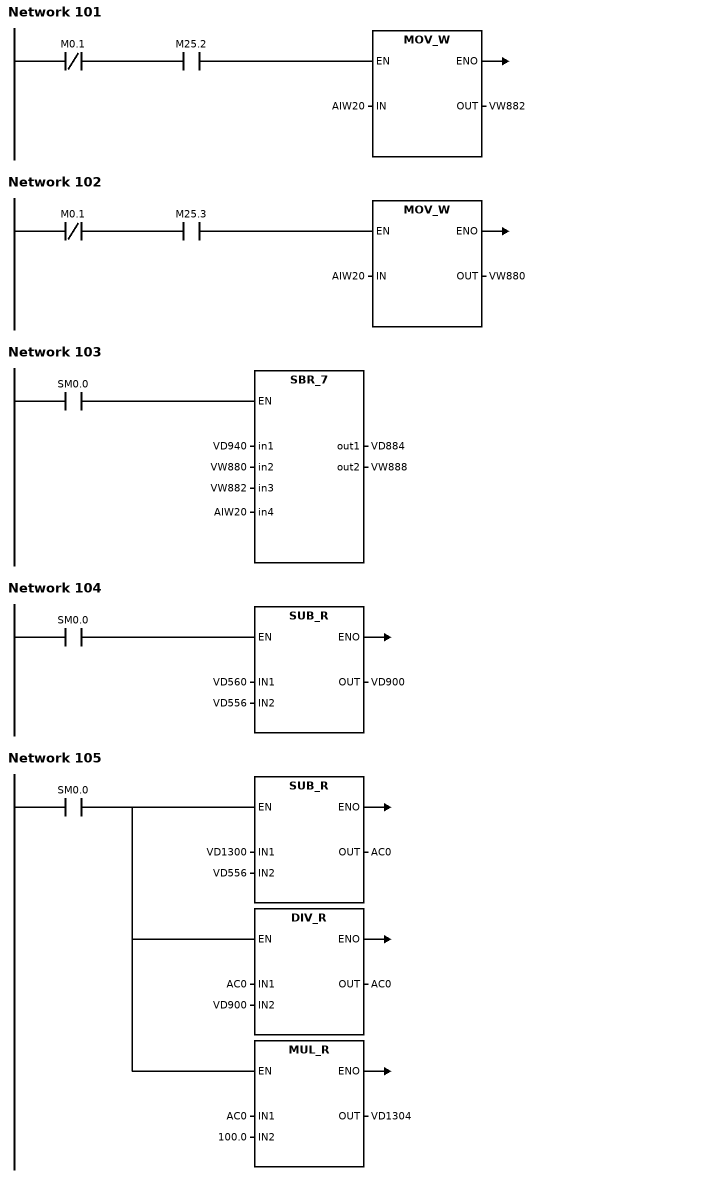
[picture p24: OB1 networks 101-105]
Network 101
LDN    M0.1
A      M25.2
MOVW   AIW20, VW882
Network 102
LDN    M0.1
A      M25.3
MOVW   AIW20, VW880
Network 103
LD     SM0.0
CALL   SBR_7:SBR7, VD940, VW880, VW882, AIW20, VD884, VW888
Network 104
LD     SM0.0
MOVR   VD560, VD900
-R     VD556, VD900
Network 105
LD     SM0.0
MOVR   VD1300, AC0
-R     VD556, AC0
/R     VD900, AC0
MOVR   AC0, VD1304
*R     100.0, VD1304
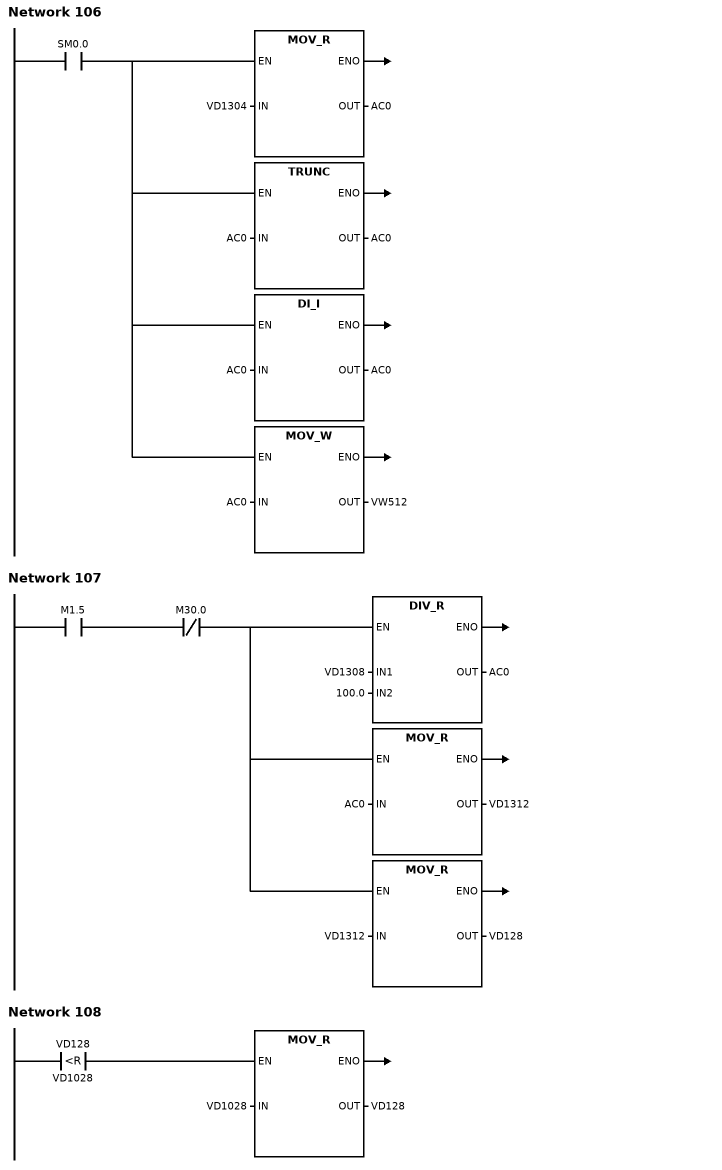
Network 106
LD     SM0.0
MOVR   VD1304, AC0
TRUNC  AC0, AC0
DTI    AC0, AC0
MOVW   AC0, VW512
Network 107
LD     M1.5
AN     M30.0
MOVR   VD1308, AC0
/R     100.0, AC0
MOVR   AC0, VD1312
MOVR   VD1312, VD128
Network 108
LDR<   VD128, VD1028
MOVR   VD1028, VD128
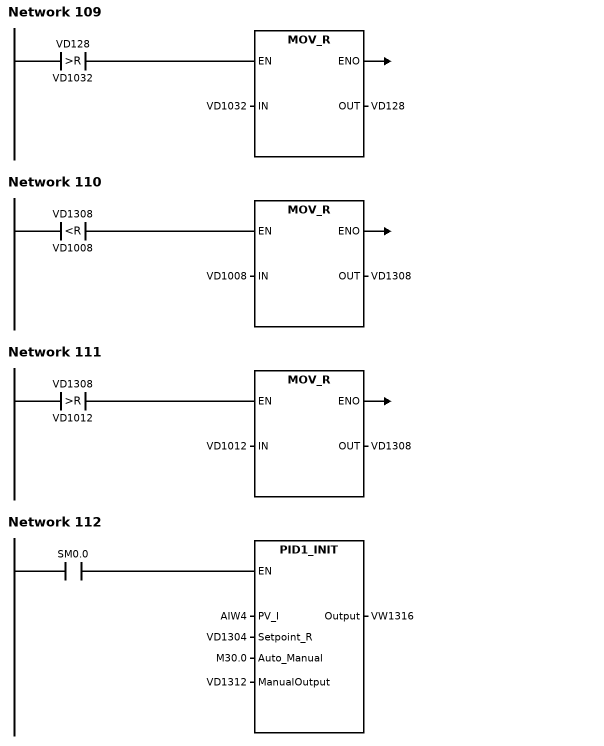
Network 109
LDR>   VD128, VD1032
MOVR   VD1032, VD128
Network 110
LDR<   VD1308, VD1008
MOVR   VD1008, VD1308
Network 111
LDR>   VD1308, VD1012
MOVR   VD1012, VD1308
Network 112
LD     SM0.0
CALL   PID1_INIT:SBR2, AIW4, VD1304, M30.0, VD1312, VW1316
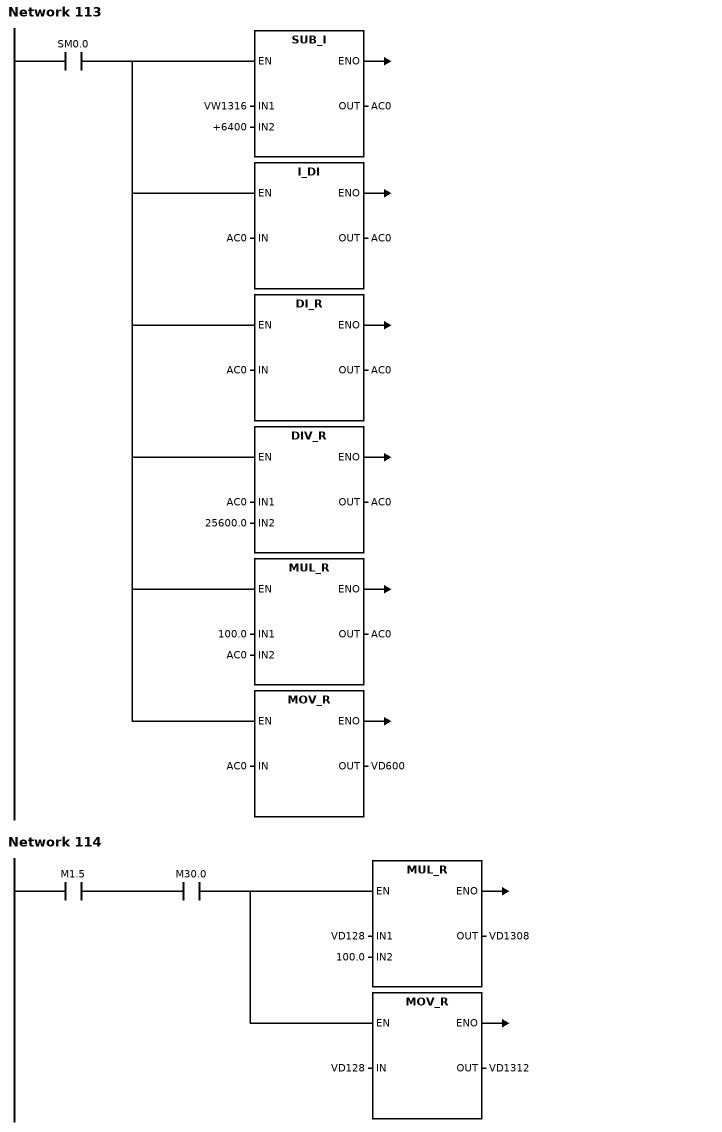
Network 113
LD     SM0.0
MOVW   VW1316, AC0
-I     +6400, AC0
ITD    AC0, AC0
DTR    AC0, AC0
/R     25600.0, AC0
*R     100.0, AC0
MOVR   AC0, VD600
Network 114
LD     M1.5
A      M30.0
MOVR   VD128, VD1308
*R     100.0, VD1308
MOVR   VD128, VD1312
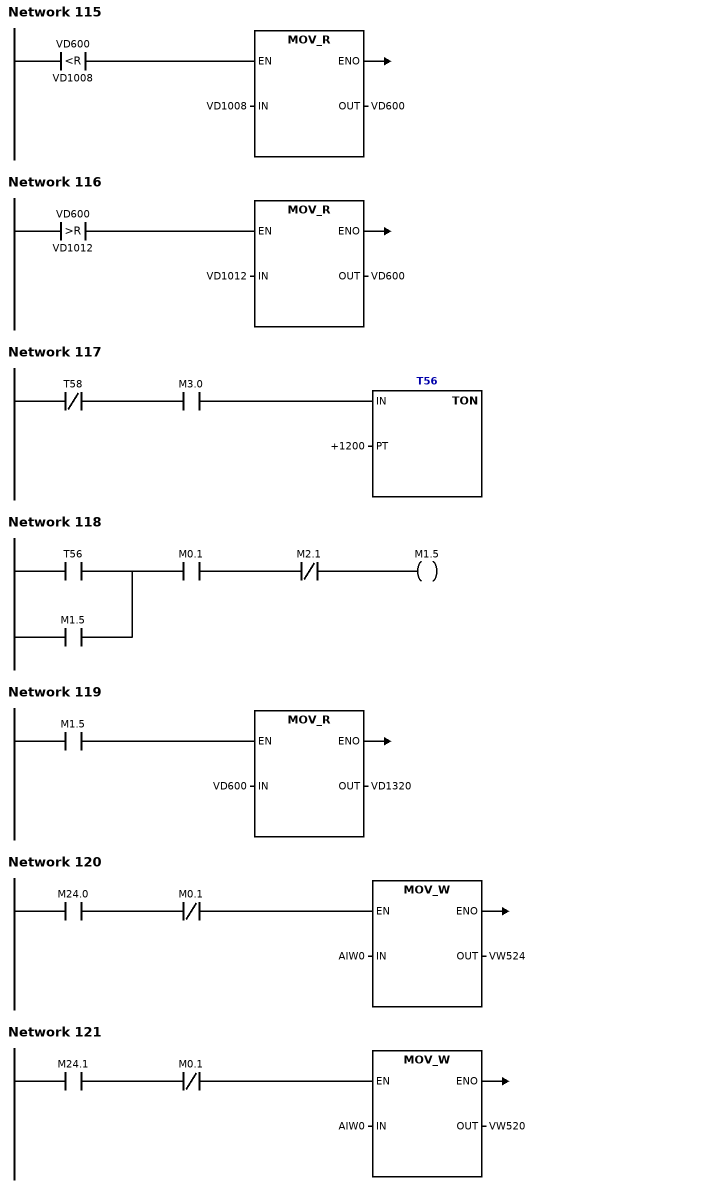
Network 115
LDR<   VD600, VD1008
MOVR   VD1008, VD600
Network 116
LDR>   VD600, VD1012
MOVR   VD1012, VD600
Network 117
LDN    T58
A      M3.0
TON    T56, +1200
Network 118
LD     T56
O      M1.5
A      M0.1
AN     M2.1
=      M1.5
Network 119
LD     M1.5
MOVR   VD600, VD1320
Network 120
LD     M24.0
AN     M0.1
MOVW   AIW0, VW524
Network 121
LD     M24.1
AN     M0.1
MOVW   AIW0, VW520
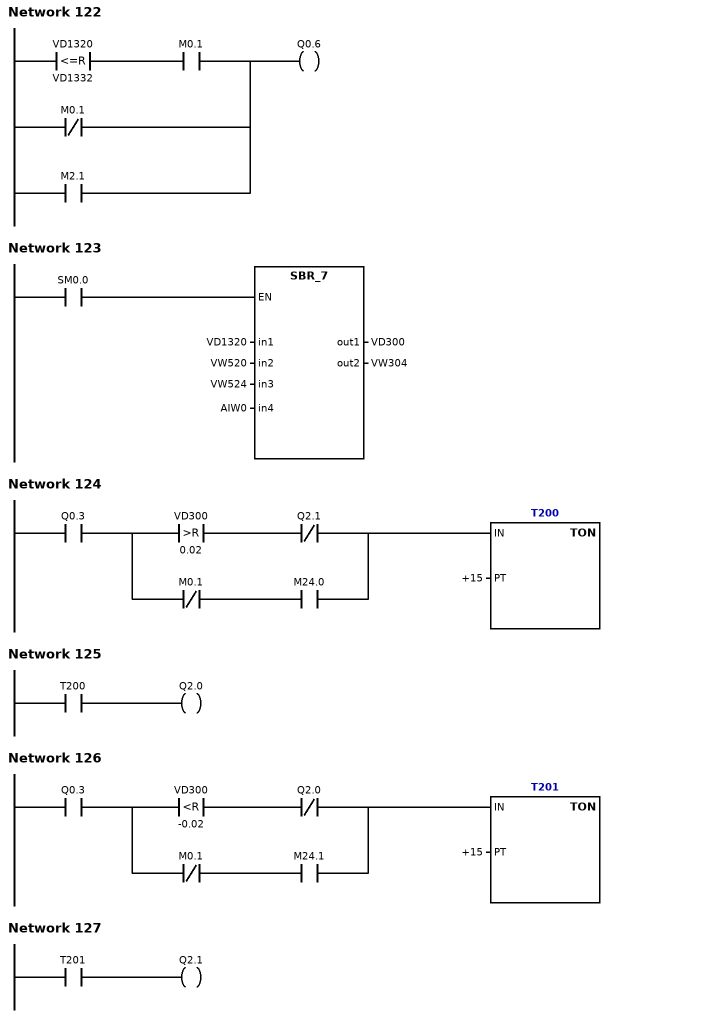
Network 122
LDR<=  VD1320, VD1332
A      M0.1
ON     M0.1
O      M2.1
=      Q0.6
Network 123
LD     SM0.0
CALL   SBR_7:SBR7, VD1320, VW520, VW524, AIW0, VD300, VW304
Network 124
LD     Q0.3
LDR>   VD300, 0.02
AN     Q2.1
LDN    M0.1
A      M24.0
OLD
ALD
TON    T200, +15
Network 125
LD     T200
=      Q2.0
Network 126
LD     Q0.3
LDR<   VD300, -0.02
AN     Q2.0
LDN    M0.1
A      M24.1
OLD
ALD
TON    T201, +15
Network 127
LD     T201
=      Q2.1
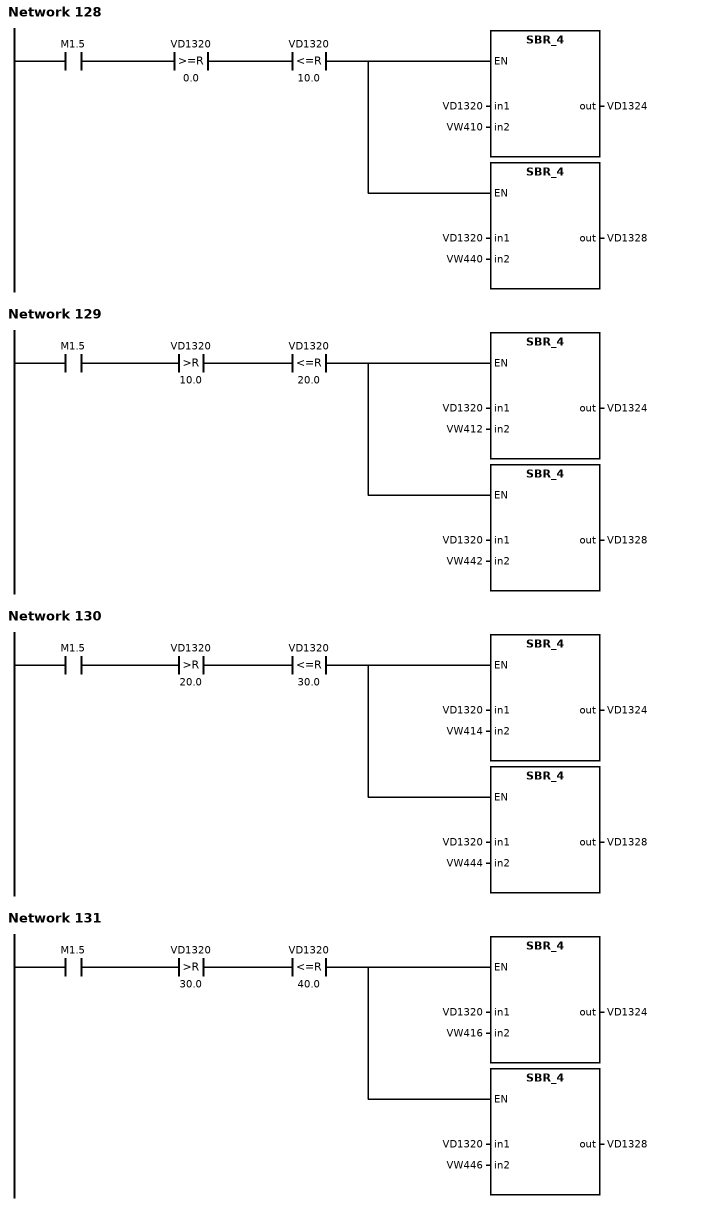
Network 128
LD     M1.5
AR>=   VD1320, 0.0
AR<=   VD1320, 10.0
CALL   SBR_4:SBR4, VD1320, VW410, VD1324
CALL   SBR_4:SBR4, VD1320, VW440, VD1328
Network 129
LD     M1.5
AR>    VD1320, 10.0
AR<=   VD1320, 20.0
CALL   SBR_4:SBR4, VD1320, VW412, VD1324
CALL   SBR_4:SBR4, VD1320, VW442, VD1328
Network 130
LD     M1.5
AR>    VD1320, 20.0
AR<=   VD1320, 30.0
CALL   SBR_4:SBR4, VD1320, VW414, VD1324
CALL   SBR_4:SBR4, VD1320, VW444, VD1328
Network 131
LD     M1.5
AR>    VD1320, 30.0
AR<=   VD1320, 40.0
CALL   SBR_4:SBR4, VD1320, VW416, VD1324
CALL   SBR_4:SBR4, VD1320, VW446, VD1328
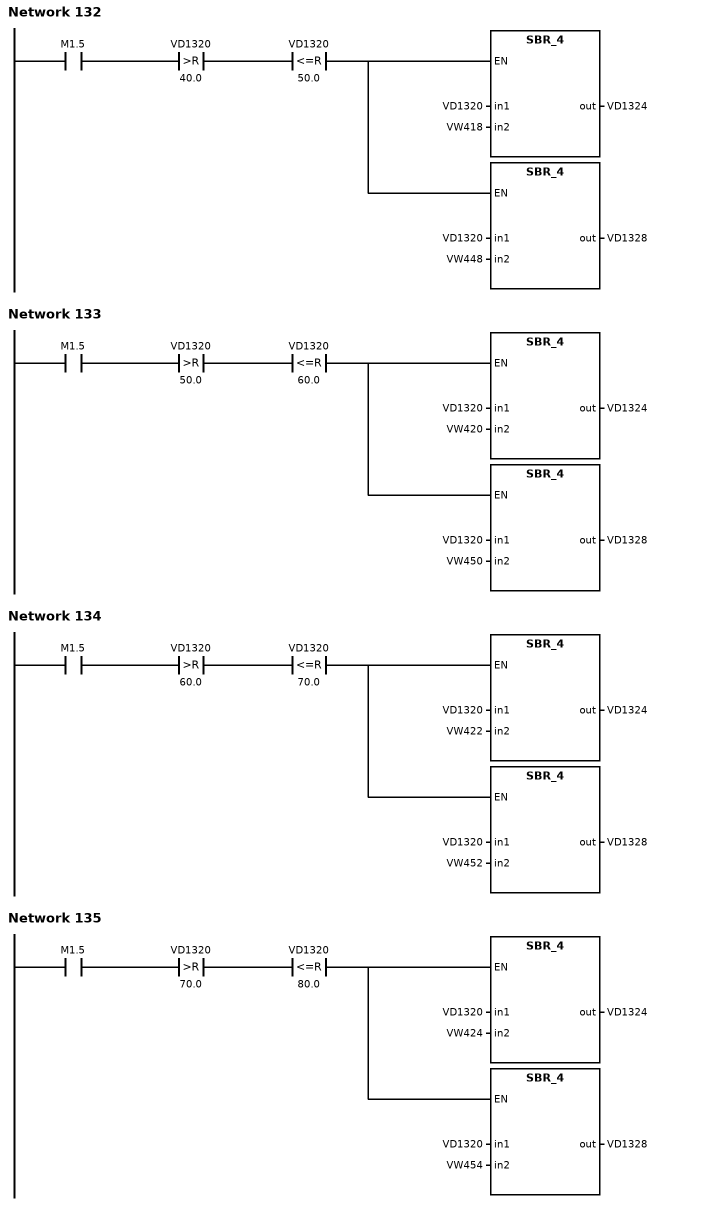
Network 132
LD     M1.5
AR>    VD1320, 40.0
AR<=   VD1320, 50.0
CALL   SBR_4:SBR4, VD1320, VW418, VD1324
CALL   SBR_4:SBR4, VD1320, VW448, VD1328
Network 133
LD     M1.5
AR>    VD1320, 50.0
AR<=   VD1320, 60.0
CALL   SBR_4:SBR4, VD1320, VW420, VD1324
CALL   SBR_4:SBR4, VD1320, VW450, VD1328
Network 134
LD     M1.5
AR>    VD1320, 60.0
AR<=   VD1320, 70.0
CALL   SBR_4:SBR4, VD1320, VW422, VD1324
CALL   SBR_4:SBR4, VD1320, VW452, VD1328
Network 135
LD     M1.5
AR>    VD1320, 70.0
AR<=   VD1320, 80.0
CALL   SBR_4:SBR4, VD1320, VW424, VD1324
CALL   SBR_4:SBR4, VD1320, VW454, VD1328
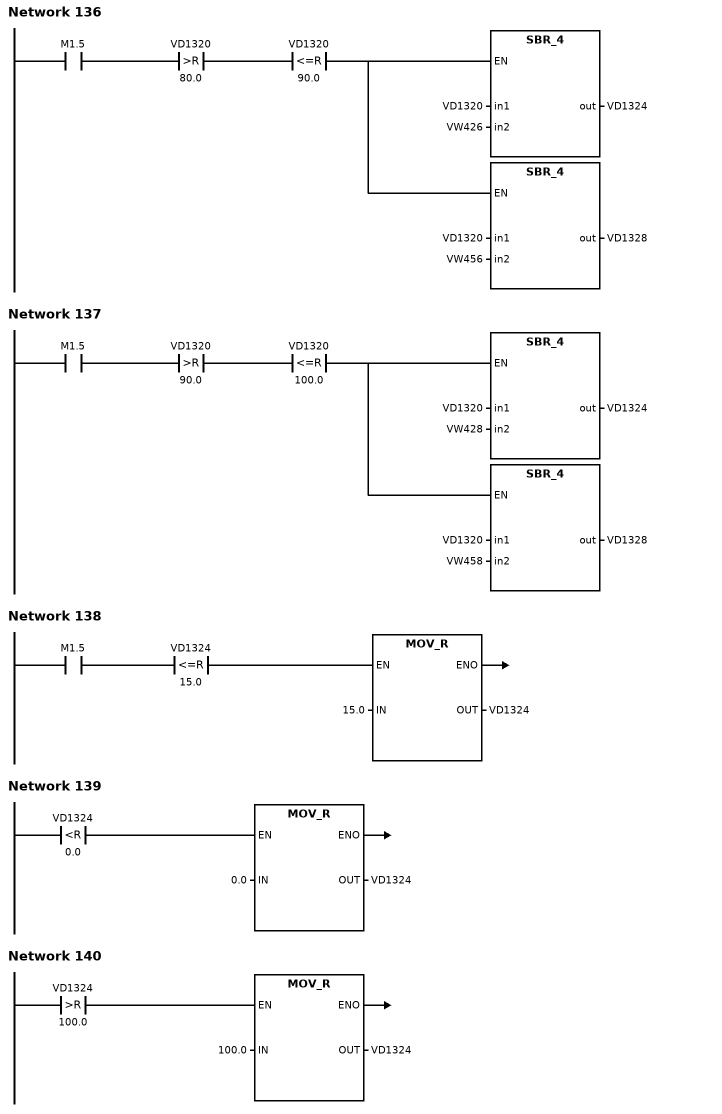
Network 136
LD     M1.5
AR>    VD1320, 80.0
AR<=   VD1320, 90.0
CALL   SBR_4:SBR4, VD1320, VW426, VD1324
CALL   SBR_4:SBR4, VD1320, VW456, VD1328
Network 137
LD     M1.5
AR>    VD1320, 90.0
AR<=   VD1320, 100.0
CALL   SBR_4:SBR4, VD1320, VW428, VD1324
CALL   SBR_4:SBR4, VD1320, VW458, VD1328
Network 138
LD     M1.5
AR<=   VD1324, 15.0
MOVR   15.0, VD1324
Network 139
LDR<   VD1324, 0.0
MOVR   0.0, VD1324
Network 140
LDR>   VD1324, 100.0
MOVR   100.0, VD1324
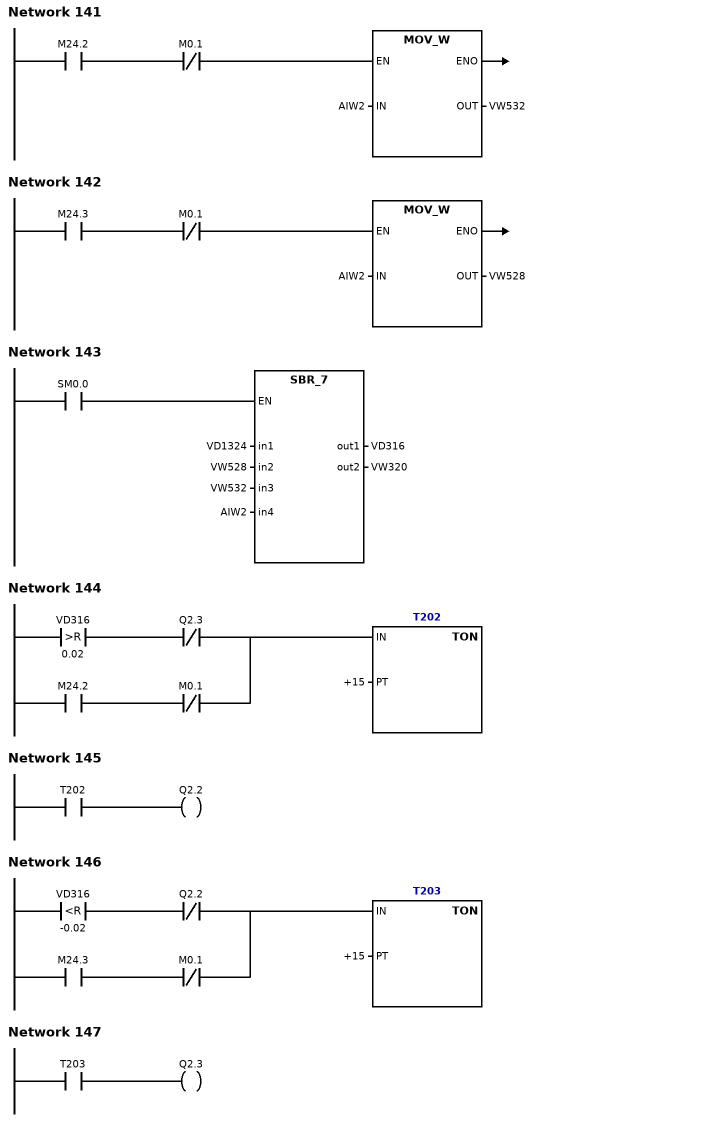
Network 141
LD     M24.2
AN     M0.1
MOVW   AIW2, VW532
Network 142
LD     M24.3
AN     M0.1
MOVW   AIW2, VW528
Network 143
LD     SM0.0
CALL   SBR_7:SBR7, VD1324, VW528, VW532, AIW2, VD316, VW320
Network 144
LDR>   VD316, 0.02
AN     Q2.3
LD     M24.2
AN     M0.1
OLD
TON    T202, +15
Network 145
LD     T202
=      Q2.2
Network 146
LDR<   VD316, -0.02
AN     Q2.2
LD     M24.3
AN     M0.1
OLD
TON    T203, +15
Network 147
LD     T203
=      Q2.3
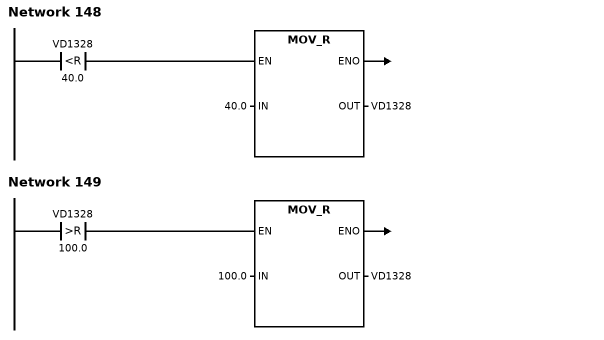
Network 148
LDR<   VD1328, 40.0
MOVR   40.0, VD1328
Network 149
LDR>   VD1328, 100.0
MOVR   100.0, VD1328
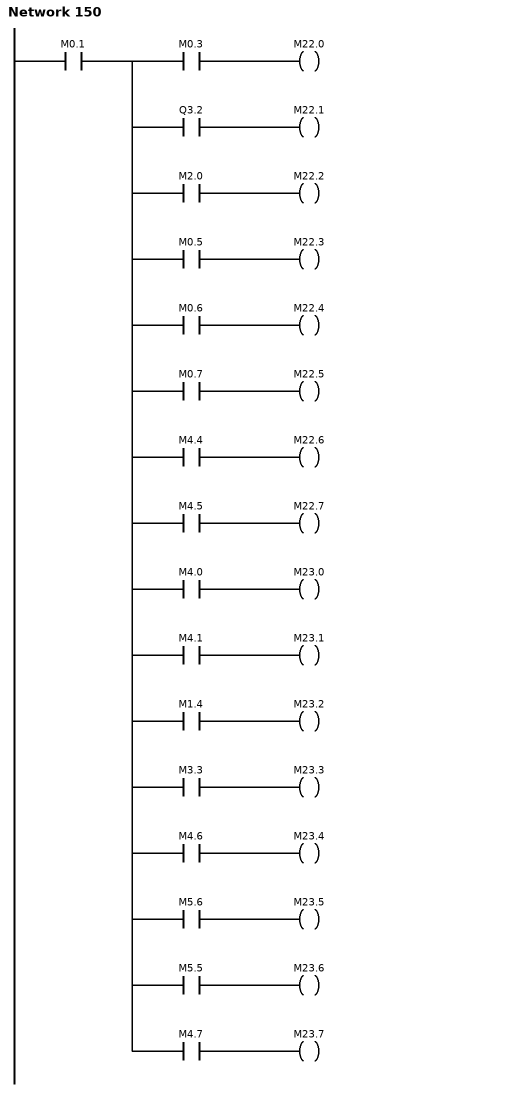
Network 150
LD     M0.1
LPS
A      M0.3
=      M22.0
LRD
A      Q3.2
=      M22.1
LRD
A      M2.0
=      M22.2
LRD
A      M0.5
=      M22.3
LRD
A      M0.6
=      M22.4
LRD
A      M0.7
=      M22.5
LRD
A      M4.4
=      M22.6
LRD
A      M4.5
=      M22.7
LRD
A      M4.0
=      M23.0
LRD
A      M4.1
=      M23.1
LRD
A      M1.4
=      M23.2
LRD
A      M3.3
=      M23.3
LRD
A      M4.6
=      M23.4
LRD
A      M5.6
=      M23.5
LRD
A      M5.5
=      M23.6
LPP
A      M4.7
=      M23.7
END_ORGANIZATION_BLOCK

// SBR1: protected block, not included

// SBR2: protected block, not included

SUBROUTINE_BLOCK SBR_3:SBR3
TITLE=
VAR_INPUT
in1:REAL;	// LD0 
in2:WORD;	// LW4 
in3:REAL;	// LD6 
END_VAR
VAR_OUTPUT
out:REAL;	// LD10 
END_VAR
BEGIN
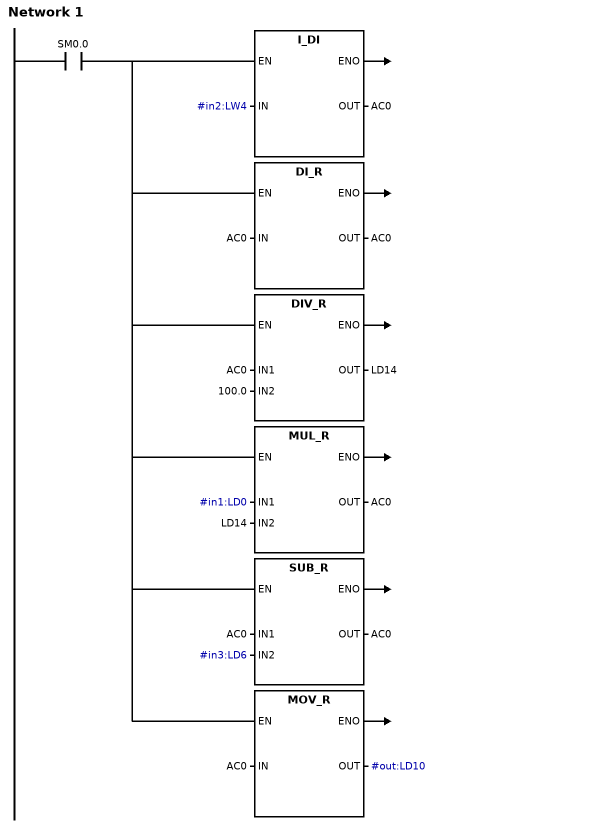
Network 1
LD     SM0.0
ITD    #in2:LW4, AC0
DTR    AC0, AC0
MOVR   AC0, LD14
/R     100.0, LD14
MOVR   #in1:LD0, AC0
*R     LD14, AC0
-R     #in3:LD6, AC0
MOVR   AC0, #out:LD10
END_SUBROUTINE_BLOCK

SUBROUTINE_BLOCK SBR_4:SBR4
TITLE=
VAR_INPUT
in1:REAL;	// LD0 
in2:WORD;	// LW4 
END_VAR
VAR_OUTPUT
out:REAL;	// LD6 
END_VAR
BEGIN
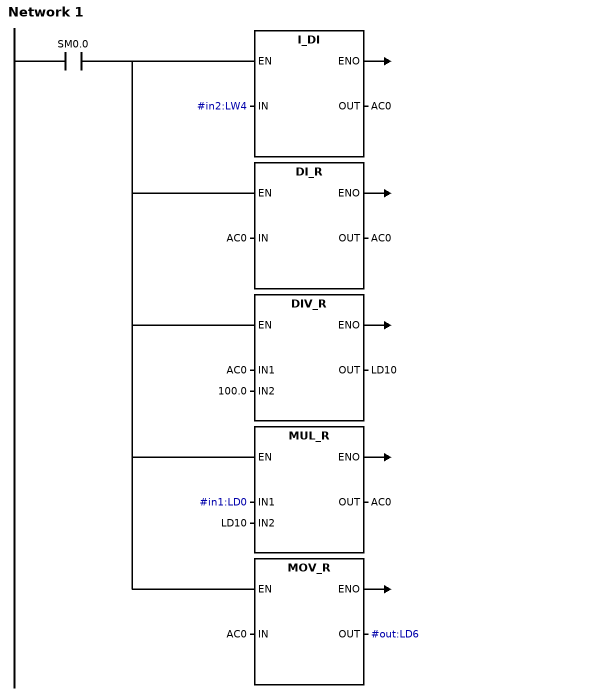
Network 1
LD     SM0.0
ITD    #in2:LW4, AC0
DTR    AC0, AC0
MOVR   AC0, LD10
/R     100.0, LD10
MOVR   #in1:LD0, AC0
*R     LD10, AC0
MOVR   AC0, #out:LD6
END_SUBROUTINE_BLOCK

SUBROUTINE_BLOCK SBR_5:SBR5
TITLE=
VAR_INPUT
zer0:REAL;	// LD0 
scan:REAL;	// LD4 
in:WORD;	// LW8 
END_VAR
VAR_OUTPUT
out:REAL;	// LD10 
END_VAR
BEGIN
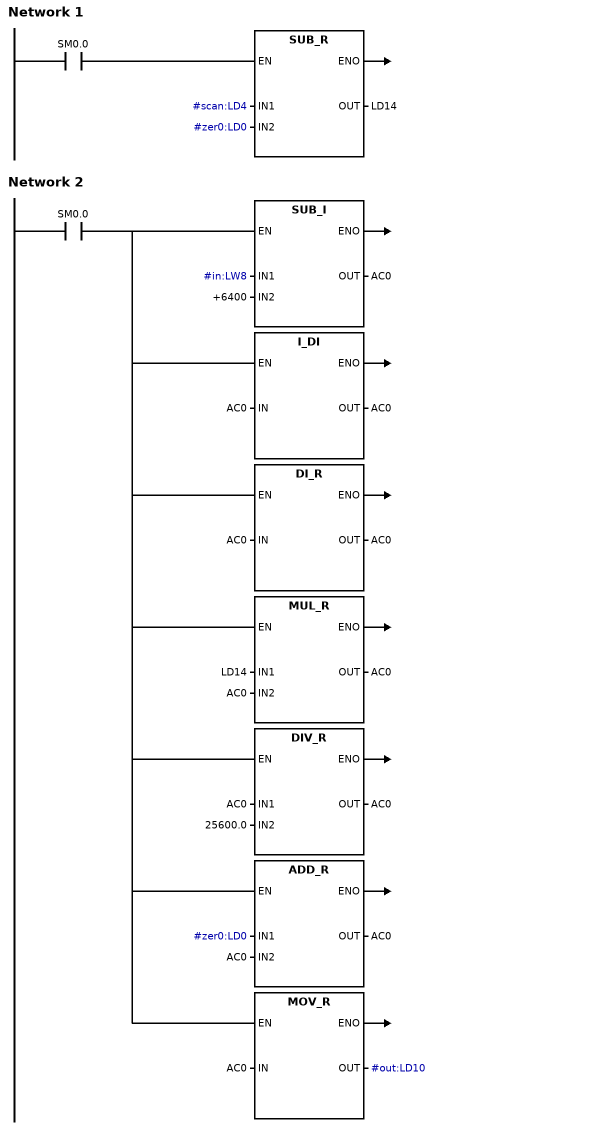
Network 1
LD     SM0.0
MOVR   #scan:LD4, LD14
-R     #zer0:LD0, LD14
Network 2
LD     SM0.0
MOVW   #in:LW8, AC0
-I     +6400, AC0
ITD    AC0, AC0
DTR    AC0, AC0
*R     LD14, AC0
/R     25600.0, AC0
+R     #zer0:LD0, AC0
MOVR   AC0, #out:LD10
END_SUBROUTINE_BLOCK

SUBROUTINE_BLOCK SBR_7:SBR7
TITLE=
VAR_INPUT
in1:REAL;	// LD0 
in2:WORD;	// LW4 
in3:WORD;	// LW6 
in4:WORD;	// LW8 
END_VAR
VAR_OUTPUT
out1:REAL;	// LD10 
out2:WORD;	// LW14 
END_VAR
BEGIN
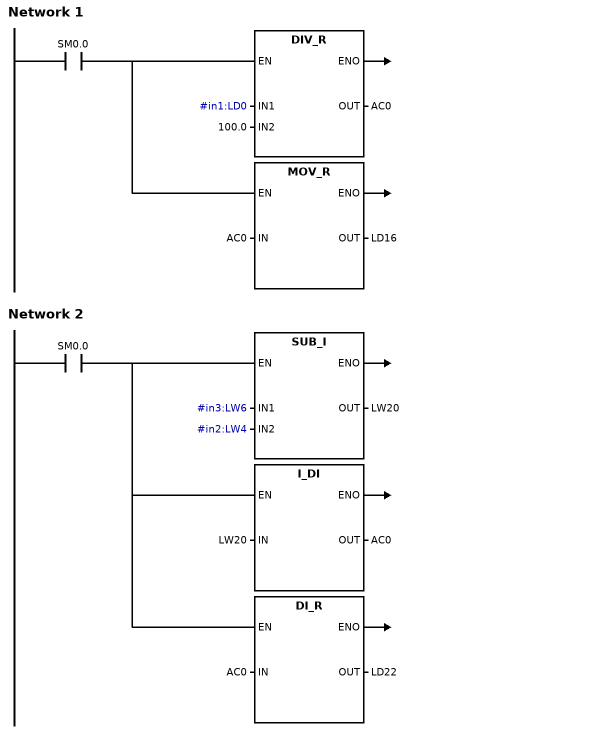
Network 1
LD     SM0.0
MOVR   #in1:LD0, AC0
/R     100.0, AC0
MOVR   AC0, LD16
Network 2
LD     SM0.0
MOVW   #in3:LW6, LW20
-I     #in2:LW4, LW20
ITD    LW20, AC0
DTR    AC0, LD22
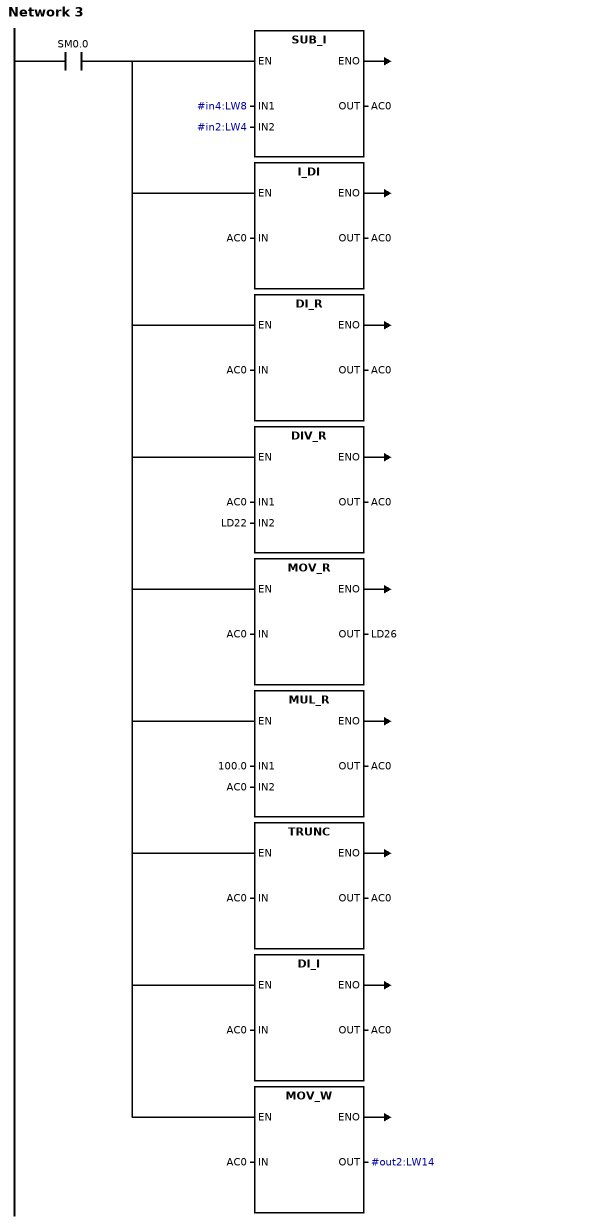
Network 3
LD     SM0.0
MOVW   #in4:LW8, AC0
-I     #in2:LW4, AC0
ITD    AC0, AC0
DTR    AC0, AC0
/R     LD22, AC0
MOVR   AC0, LD26
*R     100.0, AC0
TRUNC  AC0, AC0
DTI    AC0, AC0
MOVW   AC0, #out2:LW14
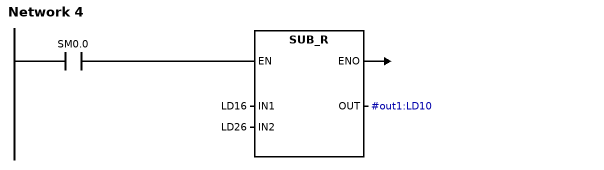
Network 4
LD     SM0.0
MOVR   LD16, #out1:LD10
-R     LD26, #out1:LD10
END_SUBROUTINE_BLOCK

// INT1: protected block, not included

// (further data pages could not be read)
